{attribute 'qualified_only'}
{attribute 'strict'}
TYPE eACRotationState :
(
	Left := -1,
	None := 0,
	Right := 1
);
END_TYPE

(* stored: Version 1.1.0.1, ProductVersion 3.1.4024.12
   DUT eACRotationState: Id {274dd091-046b-452b-a5a3-302652883fac} *)
